# B&R Automation Studio project CoffeeMachine
Automation Studio 4.1.17.113 SP; Default project

## Configuration PP400based

CPU , AutomationRuntime E3.10, Build 4.1.2, Vc V4.15.9, Safety 0.0

### Task classes (Cpu.sw)
```
Cyclic#1:
  mainlogic <- mainlogic.prg
  feeder <- FeederArm.feeder.prg
  conveyor <- ConveyorBelt.conveyor.prg
  heating <- FlowHeater.heating.prg
  brewing <- BrewingAssembly.brewing.prg
Cyclic#4:
  visCtrl <- Visualisation.visCtrl.prg
  visAlarm <- Visualisation.visAlarm.prg
  visTrend <- Visualisation.visTrend.prg
DataObjects: espres <- Recipes.espres.dob, cappu <- Recipes.cappu.dob, regular <- Recipes.regular.dob, Acp10sys, acp10sys
NcDataObjects: motor_offi <- FeederArm.motor_office.dob, motor_sim <- FeederArm.motor_sim.dob, conv_ini <- ConveyorBelt.conv_ini.dob, feed_ini <- FeederArm.feed_ini.dob, acp_err <- FeederArm.acp_err.dob
VcDataObjects: Visu <- Visualisation.Visu.dob
Binaries: vcctext, vcresman, vccovl, vcfile, vcpdpp30, vcdsloc, vcbclass, vcfntttf, vcgclass, vcshared, vcrt, vccbmp, vccbar, vcnet, vccbtn, vcmgr, vctcal, vcptelo, vcalarm, vccnum, vcdsint, Visu02, vccalarm, vcpdvnc, vcpdsw, vccline, vccstr, vcpfpp30, vcctrend, vcclbox, Visu01, vcpfmtcx, Visu03, arialbd, arial, visvc, vcchspot, arialxsr, vcchtml, vcxml, vccslider, vccurl, vccgauge, vcpkat, acp10map, acp10cfg, iomap, arconfig, asfw, sysconf, ashwd, vccshape, arialu_1, vcbmpng, vcpdcx55, vcpfpp, vcptham, ARIAL, ARIALU_1, ARIALBD, Acp10map, Acp10cfg
Libraries: powerlnk, standard, runtime, loopconr, astime, fileio, CoffeeLib, visapi, ashw, asarsdm, dataobj, Acp10_MC, brsystem, sys_lib, Acp10par, NcGlobal
```

### Hardware
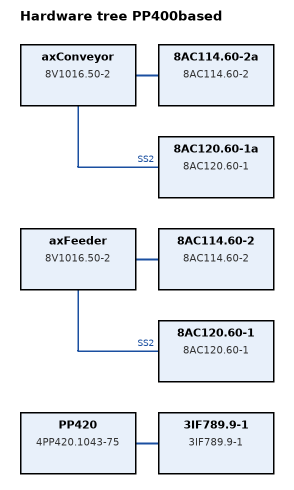
```
3IF789.9-1 : 3IF789.9-1 v1.1.1.0  [SS -> PP420.SS1]
8AC114.60-2 : 8AC114.60-2 v1.0.0.5  [SS -> axFeeder.SS1; PLK1 -> 3IF789.9-1.IF2 (NodeNumber=1)]
8AC114.60-2a : 8AC114.60-2 v1.0.0.5  [SS -> axConveyor.SS1; PLK1 -> 8AC114.60-2.PLK2 (NodeNumber=2)]
8AC120.60-1 : 8AC120.60-1 v1.0.0.2  [SS -> axFeeder.SS2]
8AC120.60-1a : 8AC120.60-1 v1.0.0.2  [SS -> axConveyor.SS2]
axConveyor : 8V1016.50-2 v1.0.0.3
axFeeder : 8V1016.50-2 v1.0.0.3
PP420 : 4PP420.1043-75 v1.0.0.0
  Connector IF5:
    ActivateDevice = 1
    Vnc1
    VncVcObjectName1 = Visu
    VncKeyMappingFile1 = PS2-Keyboard0.dis
    VncAuthentication1 = 1
    VncPasswordViewOnly1 = v
    VncPasswordViewControl1 = c
    VncRefreshRate1 = 100
    VncTitle1 = VNC - B&R Coffee Machine
  BRObjects = 460
  TimerDeviceType = EPLX2X
  TimerDevice = 3IF789.9-1.IF2
  TaskClassIdleTime = 2000
  XLinkUseDefault = 0
  XLinkDuration = 10000
  FileDevice1
  FileDeviceName1 = DISK_C
  FileDevicePath1 = C:\
  EthernetHostName = PP400CoffeeMachine
  ActivateDns = 1
  GetDnsFromDhcp = 2
  VcObjectName = Visu
```

### Acp10cfg.ncc - PP420/Motion/Acp10cfg.ncc
```
NcConfiguration (Version=2.14.0, NcSwId=acp10)
  ACP10CF1_typ:
    cnt_nettrc_rec_drive = 150
    bufsize_trace_upload = 1200
    tc_nc_man_task = Cyclic #1
    glob_pv_as_ncobject = Yes
    network_init:
      ncsw_init_execute = Yes
      automatic_execute = No
      node_nr_warning = Yes
      net_err_before_ncact = Yes
    nettrc:
      enter_parsecrec = Yes
      enter_ncaction = Yes
      save_ring_startidx = No
    plk_if[0]:
      if_name = SL1.SS1.IF2
```

### Acp10map.ncm - PP420/Motion/Acp10map.ncm
```
NcMapping (NcSwId=acp10)
  NcObject axFeeder (ModuleId=axFeeder, Type=ncAXIS, Channel=1, AcoposSimulation=Off, InitParameter=feed_ini, AcoposParameter=motor_sim, AdditionalData=PLCopen_ModPos="36000,100", Disabled=FALSE, ModuleDisabled=FALSE)
  NcObject axConveyor (ModuleId=axConveyor, Type=ncAXIS, Channel=1, AcoposSimulation=Off, InitParameter=conv_ini, AcoposParameter=motor_sim, AdditionalData=PLCopen_ModPos="8388608,100", Disabled=FALSE, ModuleDisabled=FALSE)
  NcObject SL1.SS1.IF2.ST2.VAxis1 (ModuleId=axConveyor, Type=ncV_AXIS, Channel=1, Disabled=TRUE, ModuleDisabled=FALSE)
  NcObject SL1.SS1.IF2.ST1.VAxis1 (ModuleId=axFeeder, Type=ncV_AXIS, Channel=1, Disabled=TRUE, ModuleDisabled=FALSE)
```

## Configuration PP400mcSim

CPU , AutomationRuntime E3.10, Build 4.1.2, Vc V4.15.9, Safety 0.0

### Task classes (Cpu.sw)
```
Cyclic#1 (cycle 2000 us, tolerance 0 us):
  mainlogic <- mainlogic.prg
  feeder <- FeederArm.feeder.prg
  conveyor <- ConveyorBelt.conveyor.prg
  heating <- FlowHeater.heating.prg
  brewing <- BrewingAssembly.brewing.prg
Cyclic#4 (cycle 100000 us, tolerance 100000 us):
  visCtrl <- Visualisation.visCtrl.prg
  visAlarm <- Visualisation.visAlarm.prg
  visTrend <- Visualisation.visTrend.prg
DataObjects: espres <- Recipes.espres.dob, cappu <- Recipes.cappu.dob, regular <- Recipes.regular.dob, Acp10sys
NcDataObjects: acp_err <- FeederArm.acp_err.dob, motor_sim <- FeederArm.motor_sim.dob, motor_offi <- FeederArm.motor_office.dob, conv_ini <- ConveyorBelt.conv_ini.dob, feed_ini <- FeederArm.feed_ini.dob
VcDataObjects: Visu <- Visualisation.Visu.dob
Binaries: ARIALBD, ARIALU_1, ARIAL, vcptham, vcpfpp, vcpdcx55, vcbmpng, arialu_1, vcpkat, Acp10map, Acp10cfg, vccshape, ashwd, sysconf, asfw, arconfig, iomap, acp10cfg, acp10map, vccgauge, vccslider, vccurl, vcxml, vcchtml, arialxsr, visvc, arial, arialbd, Visu03, vcpfmtcx, Visu01, vcclbox, vcctrend, vcpfpp30, vccstr, vccline, vcpdsw, vcpdvnc, vccalarm, Visu02, vcdsint, vccnum, vcalarm, vcptelo, vctcal, vcmgr, vccbtn, vcnet, vccbar, vccbmp, vcrt, vcshared, vcgclass, vcfntttf, vcbclass, vcdsloc, vcpdpp30, vcfile, vccovl, vcresman, vcctext, vcchspot
Libraries: sys_lib, brsystem, FileIO, AsTime, CoffeeLib, Acp10par, NcGlobal, AsArSdm, Acp10sdc, ashw, visapi, dataobj, loopconr, runtime, standard, powerlnk
```

### Hardware
```
PP420 : 4PP420.1043-75 v1.0.0.0
  Connector IF5:
    ActivateDevice = 1
    Vnc1
    VncVcObjectName1 = Visu
    VncAuthentication1 = 1
    VncPasswordViewOnly1 = v
    VncPasswordViewControl1 = c
    VncTitle1 = VNC - B&R Coffee Machine
  BRObjects = 450
  Cyclic1Duration = 2000
  Cyclic1Tolerance = 0
  Cyclic2Duration = 20000
  Cyclic2Tolerance = 20000
  Cyclic3Duration = 50000
  Cyclic3Tolerance = 50000
  Cyclic4Duration = 100000
  Cyclic4Tolerance = 100000
  Cyclic5Duration = 200000
  Cyclic5Tolerance = 200000
  Cyclic6Duration = 500000
  Cyclic6Tolerance = 500000
  Cyclic7Duration = 1000000
  Cyclic7Tolerance = 1000000
  Cyclic8Duration = 10000
  Cyclic8Tolerance = 30000000
  EthernetHostName = PP400CoffeeMachine
  ActivateDns = 1
  GetDnsFromDhcp = 2
  VcObjectName = Visu
```

## Configuration PP500mcSim

CPU , AutomationRuntime G4.09, Build 4.1.2, Vc V4.15.9, Safety 0.0

### Task classes (Cpu.sw)
```
Cyclic#1 (cycle 2000 us, tolerance 0 us):
  mainlogic <- mainlogic.prg
  feeder <- FeederArm.feeder.prg
  conveyor <- ConveyorBelt.conveyor.prg
  brewing <- BrewingAssembly.brewing.prg
  heating <- FlowHeater.heating.prg
Cyclic#4 (cycle 100000 us, tolerance 100000 us):
  visCtrl <- Visualisation.visCtrl.prg
  visAlarm <- Visualisation.visAlarm.prg
  visTrend <- Visualisation.visTrend.prg
DataObjects: cappu <- Recipes.cappu.dob, regular <- Recipes.regular.dob, espres <- Recipes.espres.dob, Acp10sys
NcDataObjects: acp_err <- FeederArm.acp_err.dob, motor_sim <- FeederArm.motor_sim.dob, motor_offi <- FeederArm.motor_office.dob, feed_ini <- FeederArm.feed_ini.dob, conv_ini <- ConveyorBelt.conv_ini.dob
VcDataObjects: VisuW <- Visualisation.VisuW.dob
Binaries: vccalarm, vcclbox, vcctext, vcrt, VisuW03, vccnum, vcchspot, vccbar, vccurl, vcchtml, vcfile, arialxsr, vcpdsw, vccbmp, vcshared, vcctrend, vcfntttf, vcgclass, vccovl, arialbd, vcdsint, vccslider, vcalarm, vccline, vcresman, vcdsloc, vccbtn, vccstr, vcbclass, vcxml, VisuW02, arial, vccdt, vccgauge, vcmgr, vcptelo, vcpdihd, vcpfpp50, vcpdi855, visvc, vccshape, VisuW01, vcpdi815, vcpfmtcx, vctcal, Acp10cfg, Acp10map, iomap, asfw, ashwd, sysconf, arconfig
Libraries: Acp10sdc, standard, loopconr, astime, runtime, powerlnk, CoffeeLib, Acp10par, AsArSdm, NcGlobal, brsystem, sys_lib, Acp10man, fileio, visapi, dataobj, acp10_mc
```

### Hardware
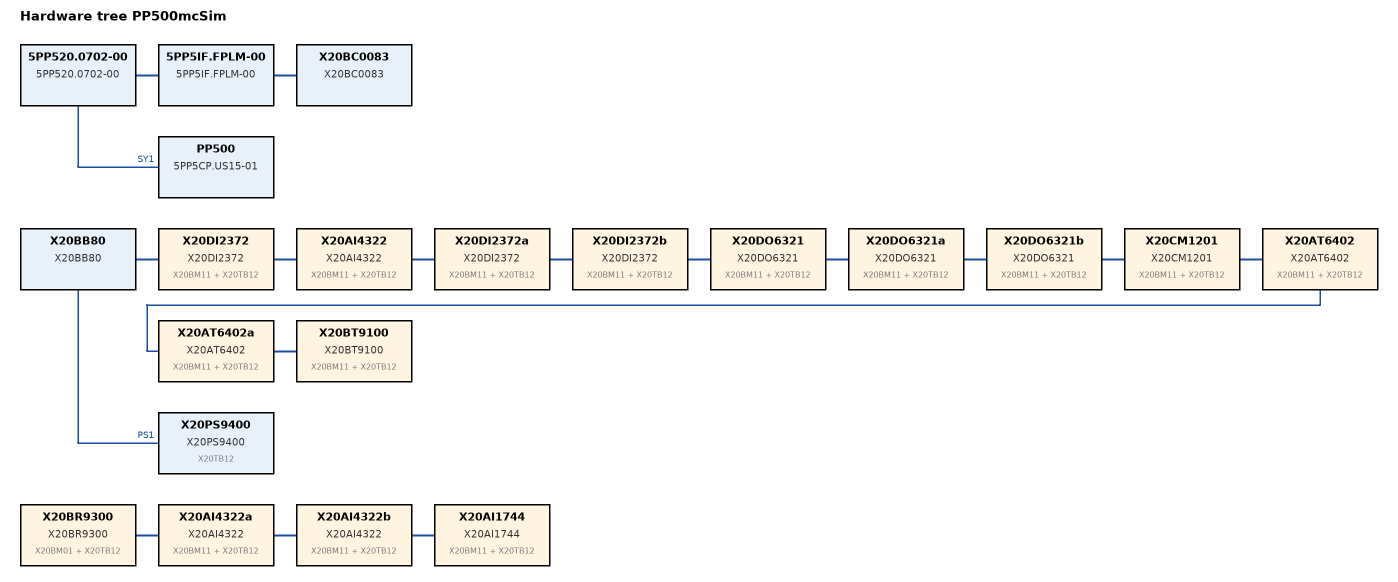
```
5PP520.0702-00 : 5PP520.0702-00 v2.0.1.2
  Connector IF3:
    ActivateDevice = 1
    EthInterfaceRedundant = 0
    HostName = pp500coffeemachine
  VcObjectName = VisuW
5PP5IF.FPLM-00 : 5PP5IF.FPLM-00 v2.2.0.0  [SL -> 5PP520.0702-00.SL1]
  Connector IF1:
    EplEthInterfaceRedundant = 0
  Supervision = off
PP500 : 5PP5CP.US15-01 v2.0.3.2  [SY -> 5PP520.0702-00.SY1]
  PreserveNonVolatileSystemSettings = 0
  BRObjects = 450
  Cyclic1Duration = 2000
  Cyclic1Tolerance = 0
  Cyclic2Duration = 20000
  Cyclic2Tolerance = 20000
  Cyclic3Duration = 50000
  Cyclic3Tolerance = 50000
  Cyclic4Duration = 100000
  Cyclic4Tolerance = 100000
  Cyclic5Duration = 200000
  Cyclic5Tolerance = 200000
  Cyclic6Duration = 500000
  Cyclic6Tolerance = 500000
  Cyclic7Duration = 1000000
  Cyclic7Tolerance = 1000000
  Cyclic8Duration = 10000
  Cyclic8Tolerance = 30000000
  EthernetHostName = brautomation
  ActivateDns = 1
X20AI1744 : X20AI1744 v1.3.0.1  [SS1 -> X20TB12o.SS; SL -> X20BM11m.SL1]
  Supervision = off
X20AI4322 : X20AI4322 v1.0.0.1  [SS1 -> X20TB12b.SS; SL -> X20BM11a.SL1]
  Supervision = off
X20AI4322a : X20AI4322 v1.0.0.1  [SS1 -> X20TB12m.SS; SL -> X20BM11k.SL1]
  Supervision = off
X20AI4322b : X20AI4322 v1.0.0.1  [SS1 -> X20TB12n.SS; SL -> X20BM11l.SL1]
  Supervision = off
X20AT6402 : X20AT6402 v1.0.2.2  [SS1 -> X20TB12i.SS; SL -> X20BM11h.SL1]
  Supervision = off
X20AT6402a : X20AT6402 v1.0.2.2  [SS1 -> X20TB12j.SS; SL -> X20BM11i.SL1]
  Supervision = off
X20BB80 : X20BB80 v1.0.0.2
X20BC0083 : X20BC0083 v2.0.0.0  [PLK1 -> 5PP5IF.FPLM-00.IF1 (NodeNumber=1); SL -> X20BB80.SL1]
  Supervision = off
X20BM01 : X20BM01 v1.0.0.1
X20BM11 : X20BM11 v1.0.0.0  [X2X1 -> X20BB80.IF1]
X20BM11a : X20BM11 v1.0.0.0  [X2X1 -> X20BM11.X2X2]
X20BM11b : X20BM11 v1.0.0.0  [X2X1 -> X20BM11a.X2X2]
X20BM11c : X20BM11 v1.0.0.0  [X2X1 -> X20BM11b.X2X2]
X20BM11d : X20BM11 v1.0.0.0  [X2X1 -> X20BM11c.X2X2]
X20BM11e : X20BM11 v1.0.0.0  [X2X1 -> X20BM11d.X2X2]
X20BM11f : X20BM11 v1.0.0.0  [X2X1 -> X20BM11e.X2X2]
X20BM11g : X20BM11 v1.0.0.0  [X2X1 -> X20BM11f.X2X2]
X20BM11h : X20BM11 v1.0.0.0  [X2X1 -> X20BM11g.X2X2]
X20BM11i : X20BM11 v1.0.0.0  [X2X1 -> X20BM11h.X2X2]
X20BM11j : X20BM11 v1.0.0.0  [X2X1 -> X20BM11i.X2X2]
X20BM11k : X20BM11 v1.0.0.0  [X2X1 -> X20BM01.X2X2]
X20BM11l : X20BM11 v1.0.0.0  [X2X1 -> X20BM11k.X2X2]
X20BM11m : X20BM11 v1.0.0.0  [X2X1 -> X20BM11l.X2X2]
X20BR9300 : X20BR9300 v1.0.2.4  [SS1 -> X20TB12l.SS; SL -> X20BM01.SL1; X2X1 -> X20BT9100.X2X1]
  Supervision = off
X20BT9100 : X20BT9100 v1.0.2.3  [SS1 -> X20TB12k.SS; SL -> X20BM11j.SL1]
  Supervision = off
X20CM1201 : X20CM1201 v1.0.0.0  [SS1 -> X20TB12h.SS; SL -> X20BM11g.SL1]
  Supervision = off
X20DI2372 : X20DI2372 v1.0.1.0  [SS1 -> X20TB12a.SS; SL -> X20BM11.SL1]
  Supervision = off
X20DI2372a : X20DI2372 v1.0.1.0  [SS1 -> X20TB12c.SS; SL -> X20BM11b.SL1]
  Supervision = off
X20DI2372b : X20DI2372 v1.0.1.0  [SS1 -> X20TB12d.SS; SL -> X20BM11c.SL1]
  Supervision = off
X20DO6321 : X20DO6321 v1.0.1.0  [SS1 -> X20TB12e.SS; SL -> X20BM11d.SL1]
  Supervision = off
X20DO6321a : X20DO6321 v1.0.1.0  [SS1 -> X20TB12f.SS; SL -> X20BM11e.SL1]
  Supervision = off
X20DO6321b : X20DO6321 v1.0.1.0  [SS1 -> X20TB12g.SS; SL -> X20BM11f.SL1]
  Supervision = off
X20PS9400 : X20PS9400 v1.0.2.0  [SS1 -> X20TB12.SS; PS -> X20BB80.PS1]
  Supervision = off
X20TB12 : X20TB12 v1.0.0.0
X20TB12a : X20TB12 v1.0.0.0
X20TB12b : X20TB12 v1.0.0.0
X20TB12c : X20TB12 v1.0.0.0
X20TB12d : X20TB12 v1.0.0.0
X20TB12e : X20TB12 v1.0.0.0
X20TB12f : X20TB12 v1.0.0.0
X20TB12g : X20TB12 v1.0.0.0
X20TB12h : X20TB12 v1.0.0.0
X20TB12i : X20TB12 v1.0.0.0
X20TB12j : X20TB12 v1.0.0.0
X20TB12k : X20TB12 v1.0.0.0
X20TB12l : X20TB12 v1.0.0.0
X20TB12m : X20TB12 v1.0.0.0
X20TB12n : X20TB12 v1.0.0.0
X20TB12o : X20TB12 v1.0.0.0
```

### Acp10cfg.ncc - PP500/Motion/Acp10cfg.ncc
```
NcConfiguration (Version=2.14.0, NcSwId=acp10)
  ACP10CF1_typ:
    cnt_nettrc_rec_drive = 150
    bufsize_trace_upload = 1200
    tc_nc_man_task = Cyclic #1
    glob_pv_as_ncobject = Yes
    network_init:
      ncsw_init_execute = Yes
      automatic_execute = No
      node_nr_warning = Yes
      net_err_before_ncact = Yes
    nettrc:
      enter_parsecrec = Yes
      enter_ncaction = Yes
    sdc_if[0]:
      if_name = SDC_IF1
```

### Acp10map.ncm - PP500/Motion/Acp10map.ncm
```
NcMapping (NcSwId=acp10)
  NcObject axFeeder (ModuleAddress=SDC_IF1.ST1, InterfaceType=SDC, Type=ncAXIS, Channel=1, AcoposSimulation=Off, InitParameter=feed_ini, AcoposParameter=motor_sim, AdditionalData=PLCopen_ModPos="36000,100", Disabled=FALSE, ModuleDisabled=FALSE)
  NcObject axConveyor (ModuleAddress=SDC_IF1.ST2, InterfaceType=SDC, Type=ncAXIS, Channel=1, AcoposSimulation=Off, InitParameter=conv_ini, AcoposParameter=motor_sim, AdditionalData=PLCopen_ModPos="8388608,100", Disabled=FALSE, ModuleDisabled=FALSE)
```

## Configuration PP65mcSim

CPU 4PP065.0571-P74, AutomationRuntime E3.10, Build 4.1.2, Vc V4.15.9, Safety 0.0

### Hardware
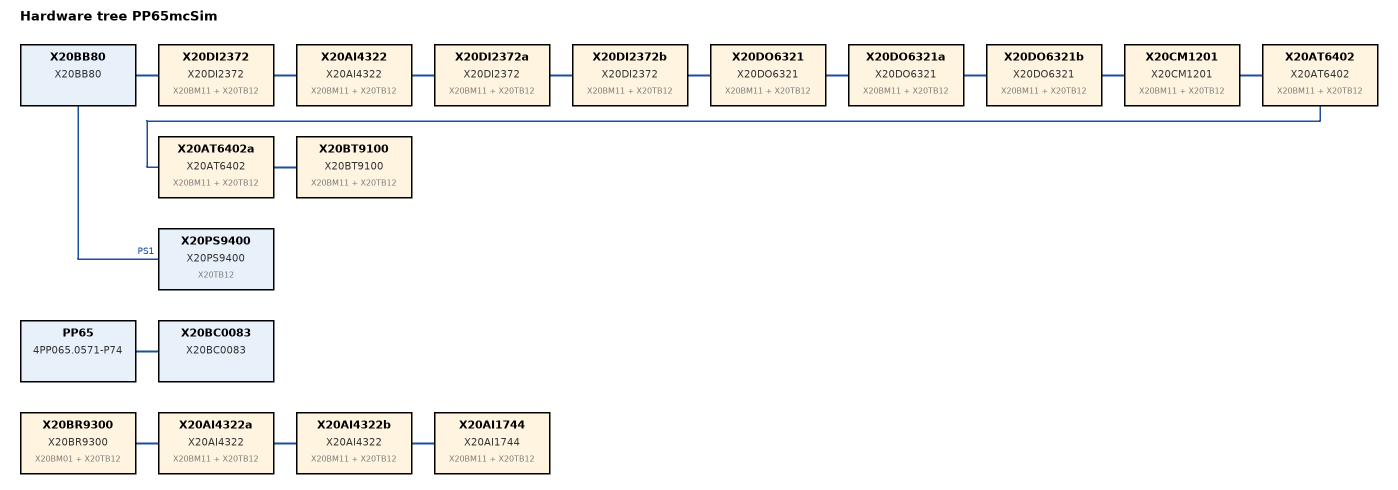
```
PP65 : 4PP065.0571-P74 v1.0.2.1
  Connector IF4:
    EplInterfaceRedundant = 0
    EplEthInterfaceRedundant = 0
  Connector IF5:
    ActivateDevice = 1
    HostName = pp500coffeemachine
    Mode = Manual
    InternetAddress = 10.49.40.222
    SubnetMask = 255.255.255.0
  PreserveNonVolatileSystemSettings = 0
  BRObjects = 450
  Cyclic1Duration = 10000
  Cyclic1Tolerance = 10000
  Cyclic2Duration = 20000
  Cyclic2Tolerance = 20000
  Cyclic3Duration = 50000
  Cyclic3Tolerance = 50000
  Cyclic4Duration = 100000
  Cyclic4Tolerance = 100000
  Cyclic5Duration = 200000
  Cyclic5Tolerance = 200000
  Cyclic6Duration = 500000
  Cyclic6Tolerance = 500000
  Cyclic7Duration = 1000000
  Cyclic7Tolerance = 1000000
  Cyclic8Duration = 10000
  Cyclic8Tolerance = 30000000
  EthernetHostName = brautomation
  ActivateDns = 1
X20AI1744 : X20AI1744 v1.3.0.1  [SS1 -> X20TB12o.SS; SL -> X20BM11m.SL1]
  Supervision = off
X20AI4322 : X20AI4322 v1.0.0.1  [SS1 -> X20TB12b.SS; SL -> X20BM11a.SL1]
  Supervision = off
X20AI4322a : X20AI4322 v1.0.0.1  [SS1 -> X20TB12m.SS; SL -> X20BM11k.SL1]
  Supervision = off
X20AI4322b : X20AI4322 v1.0.0.1  [SS1 -> X20TB12n.SS; SL -> X20BM11l.SL1]
  Supervision = off
X20AT6402 : X20AT6402 v1.0.2.2  [SS1 -> X20TB12i.SS; SL -> X20BM11h.SL1]
  Supervision = off
X20AT6402a : X20AT6402 v1.0.2.2  [SS1 -> X20TB12j.SS; SL -> X20BM11i.SL1]
  Supervision = off
X20BB80 : X20BB80 v1.0.0.2
X20BC0083 : X20BC0083 v2.0.0.0  [PLK1 -> PP65.IF4 (NodeNumber=1); SL -> X20BB80.SL1]
  Supervision = off
X20BM01 : X20BM01 v1.0.0.1
X20BM11 : X20BM11 v1.0.0.0  [X2X1 -> X20BB80.IF1]
X20BM11a : X20BM11 v1.0.0.0  [X2X1 -> X20BM11.X2X2]
X20BM11b : X20BM11 v1.0.0.0  [X2X1 -> X20BM11a.X2X2]
X20BM11c : X20BM11 v1.0.0.0  [X2X1 -> X20BM11b.X2X2]
X20BM11d : X20BM11 v1.0.0.0  [X2X1 -> X20BM11c.X2X2]
X20BM11e : X20BM11 v1.0.0.0  [X2X1 -> X20BM11d.X2X2]
X20BM11f : X20BM11 v1.0.0.0  [X2X1 -> X20BM11e.X2X2]
X20BM11g : X20BM11 v1.0.0.0  [X2X1 -> X20BM11f.X2X2]
X20BM11h : X20BM11 v1.0.0.0  [X2X1 -> X20BM11g.X2X2]
X20BM11i : X20BM11 v1.0.0.0  [X2X1 -> X20BM11h.X2X2]
X20BM11j : X20BM11 v1.0.0.0  [X2X1 -> X20BM11i.X2X2]
X20BM11k : X20BM11 v1.0.0.0  [X2X1 -> X20BM01.X2X2]
X20BM11l : X20BM11 v1.0.0.0  [X2X1 -> X20BM11k.X2X2]
X20BM11m : X20BM11 v1.0.0.0  [X2X1 -> X20BM11l.X2X2]
X20BR9300 : X20BR9300 v1.0.2.4  [SS1 -> X20TB12l.SS; SL -> X20BM01.SL1; X2X1 -> X20BT9100.X2X1]
  Supervision = off
X20BT9100 : X20BT9100 v1.0.2.3  [SS1 -> X20TB12k.SS; SL -> X20BM11j.SL1]
  Supervision = off
X20CM1201 : X20CM1201 v1.0.0.0  [SS1 -> X20TB12h.SS; SL -> X20BM11g.SL1]
  Supervision = off
X20DI2372 : X20DI2372 v1.0.1.0  [SS1 -> X20TB12a.SS; SL -> X20BM11.SL1]
  Supervision = off
X20DI2372a : X20DI2372 v1.0.1.0  [SS1 -> X20TB12c.SS; SL -> X20BM11b.SL1]
  Supervision = off
X20DI2372b : X20DI2372 v1.0.1.0  [SS1 -> X20TB12d.SS; SL -> X20BM11c.SL1]
  Supervision = off
X20DO6321 : X20DO6321 v1.0.1.2  [SS1 -> X20TB12e.SS; SL -> X20BM11d.SL1]
  Supervision = off
X20DO6321a : X20DO6321 v1.0.1.2  [SS1 -> X20TB12f.SS; SL -> X20BM11e.SL1]
  Supervision = off
X20DO6321b : X20DO6321 v1.0.1.2  [SS1 -> X20TB12g.SS; SL -> X20BM11f.SL1]
  Supervision = off
X20PS9400 : X20PS9400 v1.0.2.0  [SS1 -> X20TB12.SS; PS -> X20BB80.PS1]
  Supervision = off
X20TB12 : X20TB12 v1.0.0.0
X20TB12a : X20TB12 v1.0.0.0
X20TB12b : X20TB12 v1.0.0.0
X20TB12c : X20TB12 v1.0.0.0
X20TB12d : X20TB12 v1.0.0.0
X20TB12e : X20TB12 v1.0.0.0
X20TB12f : X20TB12 v1.0.0.0
X20TB12g : X20TB12 v1.0.0.0
X20TB12h : X20TB12 v1.0.0.0
X20TB12i : X20TB12 v1.0.0.0
X20TB12j : X20TB12 v1.0.0.0
X20TB12k : X20TB12 v1.0.0.0
X20TB12l : X20TB12 v1.0.0.0
X20TB12m : X20TB12 v1.0.0.0
X20TB12n : X20TB12 v1.0.0.0
X20TB12o : X20TB12 v1.0.0.0
```

## Configuration Simulation

CPU , AutomationRuntime G4.09, Build 4.1.2, Vc V4.15.9, Safety 0.0

### Task classes (AppMo.sw)
```
Cyclic#1 (cycle 10000 us, tolerance 0 us):
  myApptask1 <- myAppMod1.myApptask1.prg
```

### Task classes (Cpu.sw)
```
Cyclic#1 (cycle 10000 us, tolerance 0 us):
  mainlogic <- mainlogic.prg
  feeder <- FeederArm.feeder.prg
  conveyor <- ConveyorBelt.conveyor.prg
  brewing <- BrewingAssembly.brewing.prg
  heating <- FlowHeater.heating.prg
Cyclic#2:
  visCtrl <- Visualisation.visCtrl.prg
Cyclic#4:
  visAlarm <- Visualisation.visAlarm.prg
  visTrend <- Visualisation.visTrend.prg
  NewProgram <- NewProgram.prg
  myProg <- myProg.prg
DataObjects: regular <- Recipes.regular.dob, cappu <- Recipes.cappu.dob, espres <- Recipes.espres.dob, empty1 <- Recipes.empty1.dob, object2 <- Recipes.object2.dob, data <- data.dob
NcDataObjects: acp_err <- FeederArm.acp_err.dob, motor_sim <- FeederArm.motor_sim.dob, motor_offi <- FeederArm.motor_office.dob, feed_ini <- FeederArm.feed_ini.dob, conv_ini <- ConveyorBelt.conv_ini.dob, cnc1 <- cnc1.dob, cnc2 <- cnc2.dob, cnc3 <- cnc3.dob
VcDataObjects: Visu <- Visualisation.Visu.dob
Binaries: vccslider, vccurl, vcxml, vcchtml, arialxsr, vcchspot, vcctext, vcresman, vccovl, vcfile, vcdsloc, vcbclass, vcfntttf, vccstr, vcgclass, vcshared, vcrt, vccbmp, vccbar, vccbtn, vcmgr, vctcal, visvc, vcalarm, vccnum, vcdsint, vccalarm, vccline, vcpdvnc, vcpdsw, vcnet, vcctrend, vcclbox, vcpfar00, Visu01, Visu02, Visu03, vccgauge, vccshape, vccdt, arial, arialbd, acp10cfg, acp10map, arconfig, asfw, ashwd, sysconf, iomap, arialu_1, vcbmpng, ARIALU_1, Acp10map, Acp10cfg, ARIALBD, ARIAL
Libraries: AsTime, CoffeeLib, FileIO, NcGlobal, Acp10par, Convert, Visapi, AsArSdm, Runtime, operator, standard, dataobj, powerlnk, brsystem, sys_lib, Acp10man, Acp10sim, Acp10_MC, Acp10sdc, AsArProf, loopconr, vcscrsht
```

### Hardware
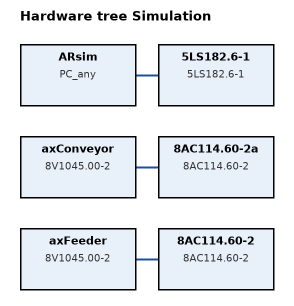
```
5LS182.6-1 : 5LS182.6-1 v1.2.2.1  [SL -> ARsim.SL1]
8AC114.60-2 : 8AC114.60-2 v1.0.0.5  [SS -> axFeeder.SS1; PLK1 -> 5LS182.6-1.IF1 (NodeNumber=1)]
8AC114.60-2a : 8AC114.60-2 v1.0.0.5  [SS -> axConveyor.SS1; PLK1 -> 8AC114.60-2.PLK2 (NodeNumber=2)]
ARsim : PC_any v1.1.0.0 (OrderNumber=PC)
  Connector IF3:
    Vnc1
    VncVcObjectName1 = Visu
    VncAuthentication1 = 1
    VncPasswordViewOnly1 = v
    VncPasswordViewControl1 = c
    VncRefreshRate1 = 200
    VncTitle1 = VNC - B&R Coffee Machine
  PreserveNonVolatileSystemSettings = 0
  BRObjects = 450
  XLinkUseDefault = 0
  Cyclic1Duration = 10000
  Cyclic1Tolerance = 0
  EthernetHostName = AR000CoffeeMachine
  ActivateOpcUa = 1
axConveyor : 8V1045.00-2 v1.0.0.2
  Simulate = standard
axFeeder : 8V1045.00-2 v1.0.0.2
  Simulate = standard
```

### Acp10cfg.ncc - ARsim/Motion/Acp10cfg.ncc
```
NcConfiguration (Version=2.37.0, NcSwId=Acp10)
  ACP10CF1_typ:
    cnt_nettrc_rec_drive = 150
    bufsize_trace_upload = 1200
    tc_nc_man_task = Cyclic #1
    glob_pv_as_ncobject = Yes
    ncsys_dl_broadcast = Yes
    ncsys_dl_acp_reset = Yes
    network_init:
      ncsw_init_execute = Yes
      automatic_execute = No
      node_nr_warning = Yes
      net_err_before_ncact = Yes
    nettrc:
      enter_parsecrec = Yes
      enter_ncaction = Yes
      save_ring_startidx = No
    plk_if[0]:
      if_name = SL1.IF1
      tc_CycDat_PLCopen = Task class for NC Manager task
      mc_broadcast_extdat = No
```

## Logical view

Binary libraries used (declarations not repeated): Convert, Runtime, sys_lib, brsystem, Standard, AsString, DataObj, FileIO, operator, AsTime, LoopConR 2.68.0, Visapi, AsArSdm, AsArProf, Acp10man 2.45.1, Acp10par 2.45.1, NcGlobal 2.45.1, Acp10sdc 2.45.1, Acp10sim 2.45.1, Acp10_MC 2.45.1

### Global.var - Global Variables
```iecst
(********************************************************************
 * COPYRIGHT -- B&R
 ********************************************************************
 * File: Global.var
 * Author: B&R
 * Created: June 06, 2007
 ********************************************************************
 * Global variables of project coffee
 ********************************************************************)
VAR
	axFeeder : ACP10AXIS_typ; (*axis information of feeder*)
	axConveyor : ACP10AXIS_typ; (*axis information of conveyor*)
	doCupPull : BOOL := FALSE; (*pulls cup out of storage*)
	gMainLogic : main_typ; (*info structure of main logic*)
	gFeeder : feeder_typ := (0); (*info structure of feeder*)
	gBrewing : brewing_typ := (0); (*info structure of brewing assembly*)
	doDoseMilk : BOOL := FALSE; (*doser: milk*)
	doDoseSugar : BOOL := FALSE; (*doser: sugar*)
	doDoseCoffee : BOOL := FALSE; (*doser: coffee*)
	gConveyor : conveyor_typ := (0);
	gHeating : heating_typ := (0); (*info structure of heating*)
	doPumpWater : BOOL := FALSE; (*water pump*)
	aoHeating : INT := 0; (*heating control*)
	atWaterTemp : INT := 0; (*actual temperature of water*)
	diStartCoffee : BOOL := FALSE; (*start making coffee*)
	gActConveyorVelocity : REAL; (*actual conveyor velocity*)
	gActFeederVelocity : REAL; (*actual feeder velocity*)
	gActFeederPosition : REAL; (*actual feeder position*)
	gActConveyorPosition : REAL; (*actual conveyor position*)
END_VAR
```

### Program Logical/mainlogic (IEC, version 1.00.0) - Main Logic Control

#### MainLogicCyclic.cfc - Cyclic code
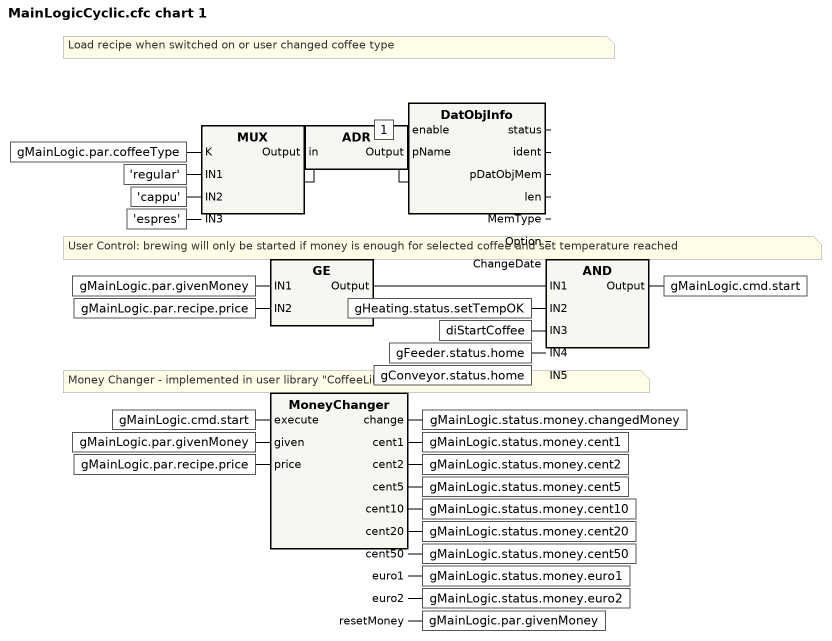
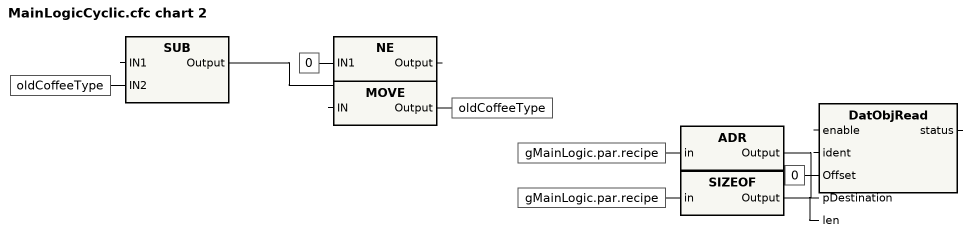
Diagram, in the editor's own instruction-list form stored in the file:
```il
PROGRAM _CYCLIC
(* Load recipe when switched on or user changed coffee type *)
(* User Control: brewing will only be started if money is enough for selected coffee and set temperature reached *)
(* Money Changer - implemented in user library "CoffeeLib" *)
VAR
	zz0000FCT_10_1_MUX_Output : ANY;
	zz0000FCT_10_1_GE_Output : BOOL;
	zz0000FB_10_1_MoneyChanger : MoneyChanger;
	zz0000FCT_10_1_ADR_Output : UDINT;
	zz0000FB_10_1_DatObjInfo : DatObjInfo;
	zz0000FCT_10_55_1_SUB_Output : ANY;
	zz0000FCT_10_55_1_NE_Output : BOOL;
	zz0000FCT_10_2_ADR_Output : UDINT;
	zz0000FCT_10_1_SIZEOF_Output : UDINT;
	zz0000FB_10_1_DatObjRead : DatObjRead;
END_VAR

LD gMainLogic.par.coffeeType
MUX 'regular', 'cappu', 'espres'
ST zz0000FCT_10_1_MUX_Output
LD gMainLogic.par.givenMoney
GE gMainLogic.par.recipe.price
ST zz0000FCT_10_1_GE_Output
LD gMainLogic.cmd.start
ST zz0000FB_10_1_MoneyChanger.execute
LD gMainLogic.par.givenMoney
ST zz0000FB_10_1_MoneyChanger.given
LD gMainLogic.par.recipe.price
ST zz0000FB_10_1_MoneyChanger.price
CAL zz0000FB_10_1_MoneyChanger
LD zz0000FB_10_1_MoneyChanger.change
ST gMainLogic.status.money.changedMoney
LD zz0000FB_10_1_MoneyChanger.cent1
ST gMainLogic.status.money.cent1
LD zz0000FB_10_1_MoneyChanger.cent2
ST gMainLogic.status.money.cent2
LD zz0000FB_10_1_MoneyChanger.cent5
ST gMainLogic.status.money.cent5
LD zz0000FB_10_1_MoneyChanger.cent10
ST gMainLogic.status.money.cent10
LD zz0000FB_10_1_MoneyChanger.cent20
ST gMainLogic.status.money.cent20
LD zz0000FB_10_1_MoneyChanger.cent50
ST gMainLogic.status.money.cent50
LD zz0000FB_10_1_MoneyChanger.euro1
ST gMainLogic.status.money.euro1
LD zz0000FB_10_1_MoneyChanger.euro2
ST gMainLogic.status.money.euro2
LD zz0000FB_10_1_MoneyChanger.resetMoney
ST gMainLogic.par.givenMoney
LD zz0000FCT_10_1_MUX_Output
ADR
ST zz0000FCT_10_1_ADR_Output
LD 1
ST zz0000FB_10_1_DatObjInfo.enable
LD zz0000FCT_10_1_ADR_Output
ST zz0000FB_10_1_DatObjInfo.pName
CAL zz0000FB_10_1_DatObjInfo
LD zz0000FCT_10_1_GE_Output
AND gHeating.status.setTempOK
AND diStartCoffee
AND gFeeder.status.home
AND gConveyor.status.home
ST gMainLogic.cmd.start
LD gMainLogic.par.coffeeType
SUB oldCoffeeType
ST zz0000FCT_10_55_1_SUB_Output
LD 0
NE zz0000FCT_10_55_1_SUB_Output
ST zz0000FCT_10_55_1_NE_Output
LD gMainLogic.par.coffeeType
MOVE
ST oldCoffeeType
LD gMainLogic.par.recipe
ADR
ST zz0000FCT_10_2_ADR_Output
LD gMainLogic.par.recipe
SIZEOF
ST zz0000FCT_10_1_SIZEOF_Output
LD zz0000FCT_10_55_1_NE_Output
ST zz0000FB_10_1_DatObjRead.enable
LD zz0000FB_10_1_DatObjInfo.ident
ST zz0000FB_10_1_DatObjRead.ident
LD 0
ST zz0000FB_10_1_DatObjRead.Offset
LD zz0000FCT_10_2_ADR_Output
ST zz0000FB_10_1_DatObjRead.pDestination
LD zz0000FCT_10_1_SIZEOF_Output
ST zz0000FB_10_1_DatObjRead.len
CAL zz0000FB_10_1_DatObjRead

END_PROGRAM
```

#### MainLogicInit.cfc
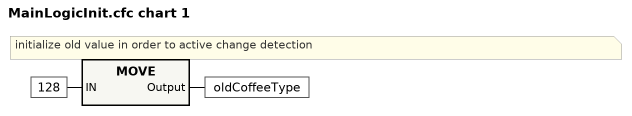
Diagram, in the editor's own instruction-list form stored in the file:
```il
PROGRAM _INIT
(* initialize old value in order to active change detection *)

LD  128
MOVE
ST oldCoffeeType

END_PROGRAM
```

#### mainlogic.var - Local variables
```iecst
(********************************************************************
 * COPYRIGHT -- B&R
 ********************************************************************
 * Package: mainlogic
 * File: mainlogic.var
 * Author: B&R
 * Created: June 18, 2007
 *******************************************************************)
VAR
	oldCoffeeType : SINT := 0;
END_VAR
```

### Package Logical/ConveyorBelt - Conveyor Control

### Data object Logical/ConveyorBelt/conv_ini (Ax) - Conveyor axis configuration

#### conv_ini.ax
```
InitParameter (Version=2.28.2, NcSwId=ACP10)
  ACP10AXIS_typ:
    dig_in:
      level:
        reference = ncACTIV_HI
        pos_hw_end = ncACTIV_HI
        neg_hw_end = ncACTIV_HI
        trigger1 = ncACTIV_HI
        trigger2 = ncACTIV_HI
    encoder_if:
      parameter:
        count_dir = ncSTANDARD
        scaling:
          load:
            units = 5000
            rev_motor = 10
    limit:
      parameter:
        v_pos = 10000
        v_neg = 10000
        a1_pos = 50000
        a2_pos = 50000
        a1_neg = 50000
        a2_neg = 50000
        t_jolt = 0.05
        t_in_pos = 0
        pos_sw_end = 8388607
        neg_sw_end = -8388608
        ds_warning = 500
        ds_stop = 1000
        a_stop = 1e+030
        dv_stop = 0
        dv_stop_mode = ncOFF
    controller:
      mode = ncPOSITION
      position:
        kv = 50
        tn = 0
        t_predict = 0.0008
        t_total = 0.0008
        p_max = 10000
        i_max = 0
      speed:
        kv = 2
        tn = 0
        t_filter = 0
        isq_filter1:
          type = ncOFF
          a0 = 0
          a1 = 0
          b0 = 0
          b1 = 0
          b2 = 0
          c0_par_id = 0
          c1_par_id = 0
        isq_filter2:
          type = ncOFF
          a0 = 0
          a1 = 0
          b0 = 0
          b1 = 0
          b2 = 0
          c0_par_id = 0
          c1_par_id = 0
        isq_filter3:
          type = ncOFF
          a0 = 0
          a1 = 0
          b0 = 0
          b1 = 0
          b2 = 0
          c0_par_id = 0
          c1_par_id = 0
      uf:
        type = ncLINEAR
        auto_config = ncMOTOR_PAR
        u0 = 0
        un = 0
        fn = 50
        k_f_slip = 0
      ff:
        torque_load = 0
        torque_pos = 0
        torque_neg = 0
        kv_torque = 0
        inertia = 0
        t_filter_a = 0
    move:
      stop:
        parameter[0]:
          decel_ramp = ncA_LIMIT
          controller = ncON
        parameter[1]:
          decel_ramp = ncA_LIMIT
          controller = ncON
        parameter[2]:
          decel_ramp = ncA_LIMIT
          controller = ncON
        parameter[3]:
          decel_ramp = ncA_LIMIT
          controller = ncON
        quickstop:
          decel_ramp = ncA_LIMIT
        drive_error:
          decel_ramp = ncA_LIMIT
      homing:
        parameter:
          s = 0
          v_switch = 5000
          v_trigger = 500
          a = 50000
          mode = ncDIRECT
          edge_sw = ncPOSITIVE
          start_dir = ncPOSITIVE
          trigg_dir = ncPOSITIVE
          ref_pulse = ncOFF
          tr_s_block = 0
      basis:
        parameter:
          v_pos = 10000
          v_neg = 10000
          a1_pos = 50000
          a2_pos = 50000
          a1_neg = 50000
          a2_neg = 50000
    message:
      text:
        parameter:
          format = ncBREAK
          columns = 80
          data_modul = acp_err
```

### Program Logical/ConveyorBelt/conveyor (IEC) - Conveyor Logic Control

#### conveyorCyclic.ld - Cyclic code
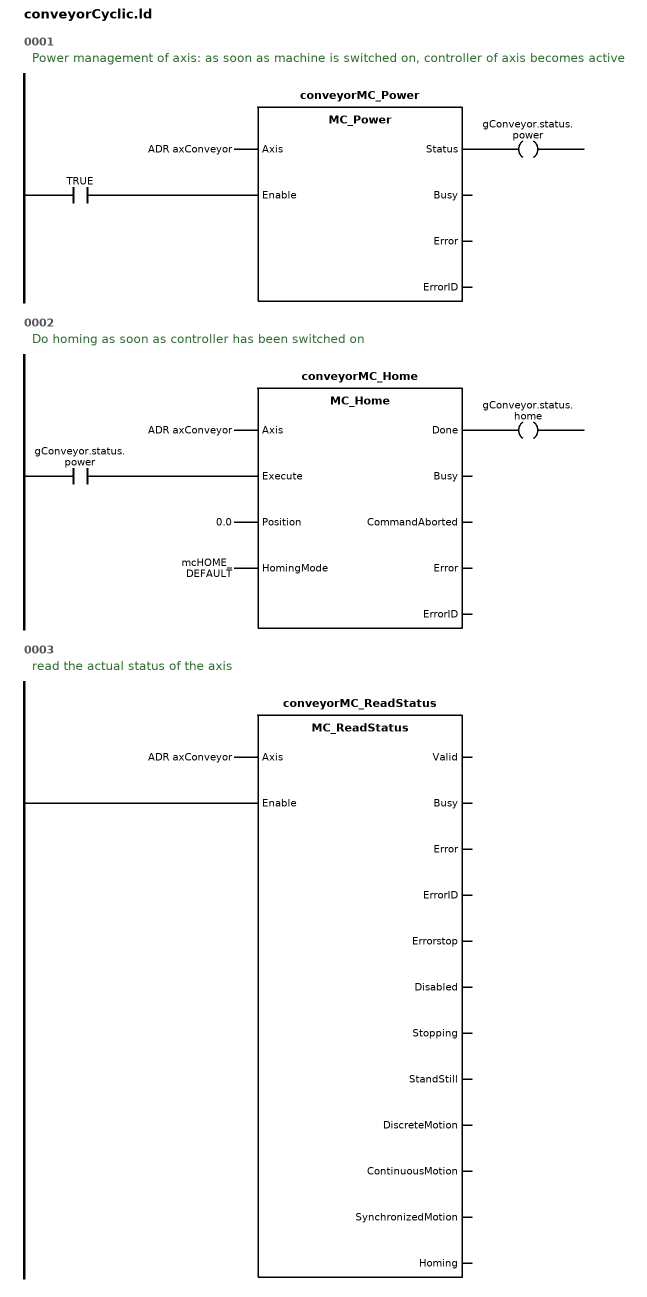
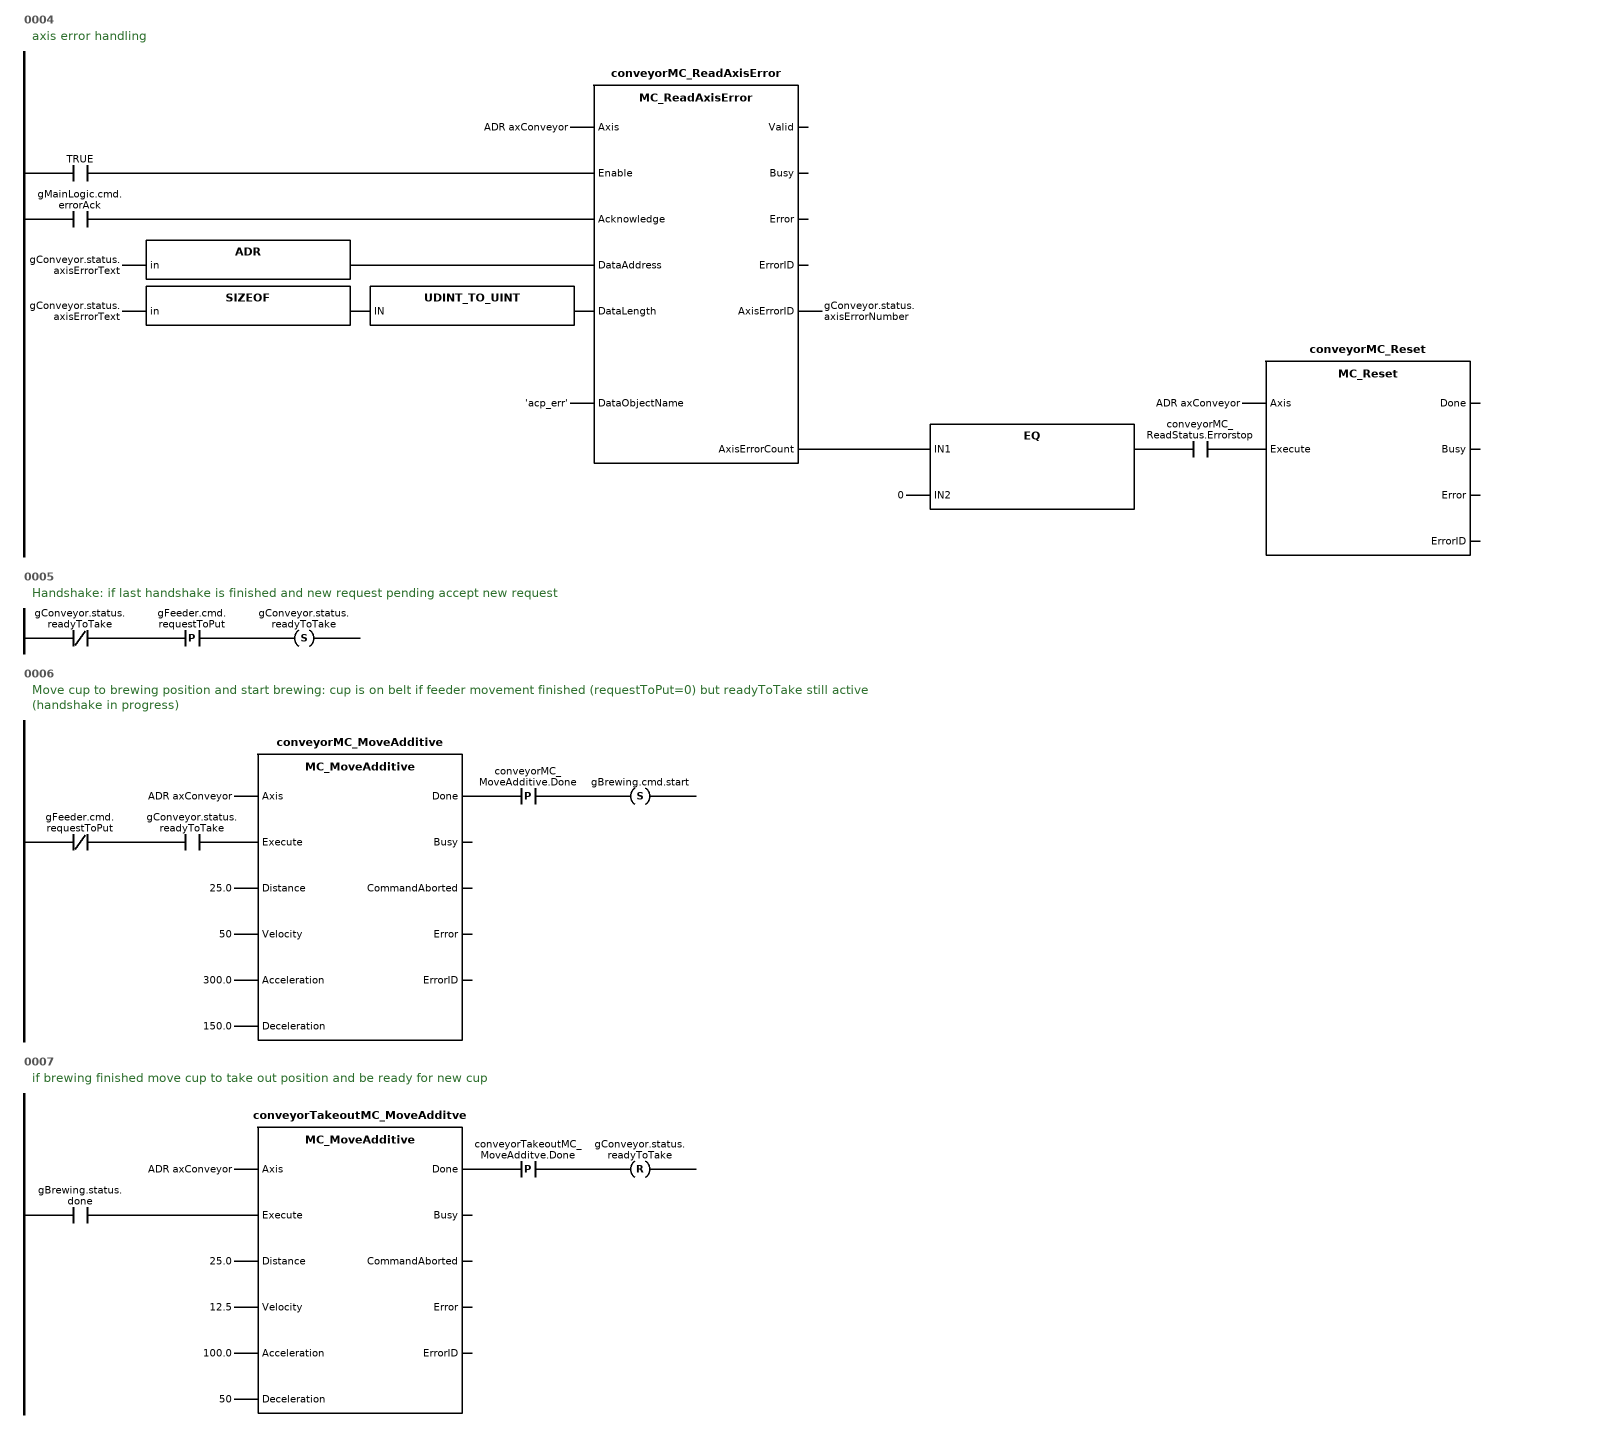
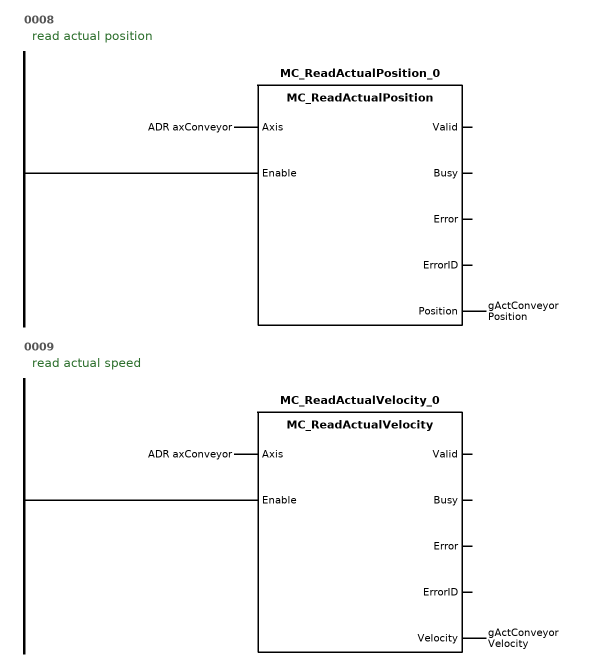
Ladder, written as Structured Text:
```iecst
(********************************************************************
 * COPYRIGHT -- Bernecker + Rainer
 ********************************************************************
 * Program: conveyor
 * File: conveyorCyclic.ld
 * Author: paulinw
 * Created: June 12, 2007
 ********************************************************************
 * Implementation of program conveyor
 ********************************************************************)

PROGRAM _CYCLIC
VAR
    _e1 : R_TRIG;
    _e2 : R_TRIG;
    _e3 : R_TRIG;
END_VAR
(* Network 1: Power management of axis: as soon as machine is switched on, controller of axis becomes active *)
conveyorMC_Power(Axis := ADR(axConveyor), Enable := TRUE);
gConveyor.status.power := conveyorMC_Power.Status;

(* Network 2: Do homing as soon as controller has been switched on *)
conveyorMC_Home(Axis := ADR(axConveyor), Execute := gConveyor.status.power, Position := 0.0, HomingMode := mcHOME_DEFAULT);
gConveyor.status.home := conveyorMC_Home.Done;

(* Network 3: read the actual status of the axis *)
conveyorMC_ReadStatus(Axis := ADR(axConveyor), Enable := TRUE);

(* Network 4: axis error handling *)
conveyorMC_ReadAxisError(Axis := ADR(axConveyor), Enable := TRUE, Acknowledge := gMainLogic.cmd.errorAck, DataAddress := ADR(in := gConveyor.status.axisErrorText), DataLength := UDINT_TO_UINT(SIZEOF(in := gConveyor.status.axisErrorText)), DataObjectName := 'acp_err');
gConveyor.status.axisErrorNumber := conveyorMC_ReadAxisError.AxisErrorID;
conveyorMC_Reset(Axis := ADR(axConveyor), Execute := (conveyorMC_ReadAxisError.AxisErrorCount = 0) AND conveyorMC_ReadStatus.Errorstop);

(* Network 5: Handshake: if last handshake is finished and new request pending accept new request *)
_e1(CLK := gFeeder.cmd.requestToPut);
IF NOT gConveyor.status.readyToTake AND _e1.Q THEN gConveyor.status.readyToTake := TRUE; END_IF;

(* Network 6: Move cup to brewing position and start brewing: cup is on belt if feeder movement finished (requestToPut=0) but readyToTake still active (handshake in progress) *)
conveyorMC_MoveAdditive(Axis := ADR(axConveyor), Execute := NOT gFeeder.cmd.requestToPut AND gConveyor.status.readyToTake, Distance := 25.0, Velocity := 50, Acceleration := 300.0, Deceleration := 150.0);
_e2(CLK := conveyorMC_MoveAdditive.Done);
IF conveyorMC_MoveAdditive.Done AND _e2.Q THEN gBrewing.cmd.start := TRUE; END_IF;

(* Network 7: if brewing finished move cup to take out position and be ready for new cup *)
conveyorTakeoutMC_MoveAdditve(Axis := ADR(axConveyor), Execute := gBrewing.status.done, Distance := 25.0, Velocity := 12.5, Acceleration := 100.0, Deceleration := 50);
_e3(CLK := conveyorTakeoutMC_MoveAdditve.Done);
IF conveyorTakeoutMC_MoveAdditve.Done AND _e3.Q THEN gConveyor.status.readyToTake := FALSE; END_IF;

(* Network 8: read actual position  *)
MC_ReadActualPosition_0(Axis := ADR(axConveyor), Enable := TRUE);
gActConveyorPosition := MC_ReadActualPosition_0.Position;

(* Network 9: read actual speed *)
MC_ReadActualVelocity_0(Axis := ADR(axConveyor), Enable := TRUE);
gActConveyorVelocity := MC_ReadActualVelocity_0.Velocity;
END_PROGRAM
```

### Package Logical/BrewingAssembly - Brewing & Dosing

### Program Logical/BrewingAssembly/brewing (IEC)

#### brewing.var - Local variables
```iecst
(********************************************************************
 * COPYRIGHT -- B&R
 ********************************************************************
 * Package: Brewing
 * File: brewing.var
 * Author: B&R
 * Created: June 14, 2007
 *******************************************************************)
VAR
	pBrewingText : UDINT := 0;
END_VAR
VAR CONSTANT
	sSTANDBY : UINT := 0;
	sDOSING : UINT := 10;
	sBREWING : UINT := 20;
	sFINISH : UINT := 30;
END_VAR
VAR
	milkTP : TP;
	coffeeTP : TP;
	sugarTP : TP;
	waterTP : TP;
END_VAR
```

### Package Logical/FeederArm - Feeder Control

### Data object Logical/FeederArm/acp_err (Ett)

- acp_err.ett (not shown)

- Data object Logical/FeederArm/feed_ini (Ax) (no source held here)

### Program Logical/FeederArm/feeder (IEC)

#### feederCyclic.ld - Cyclic code
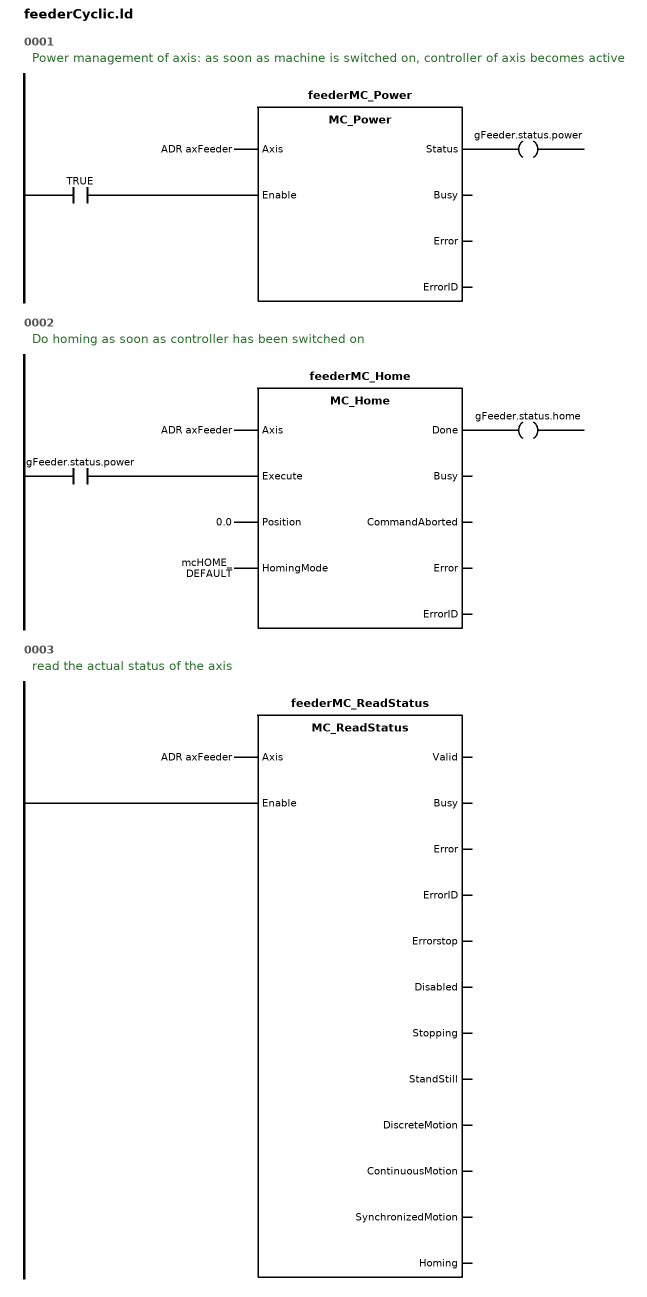
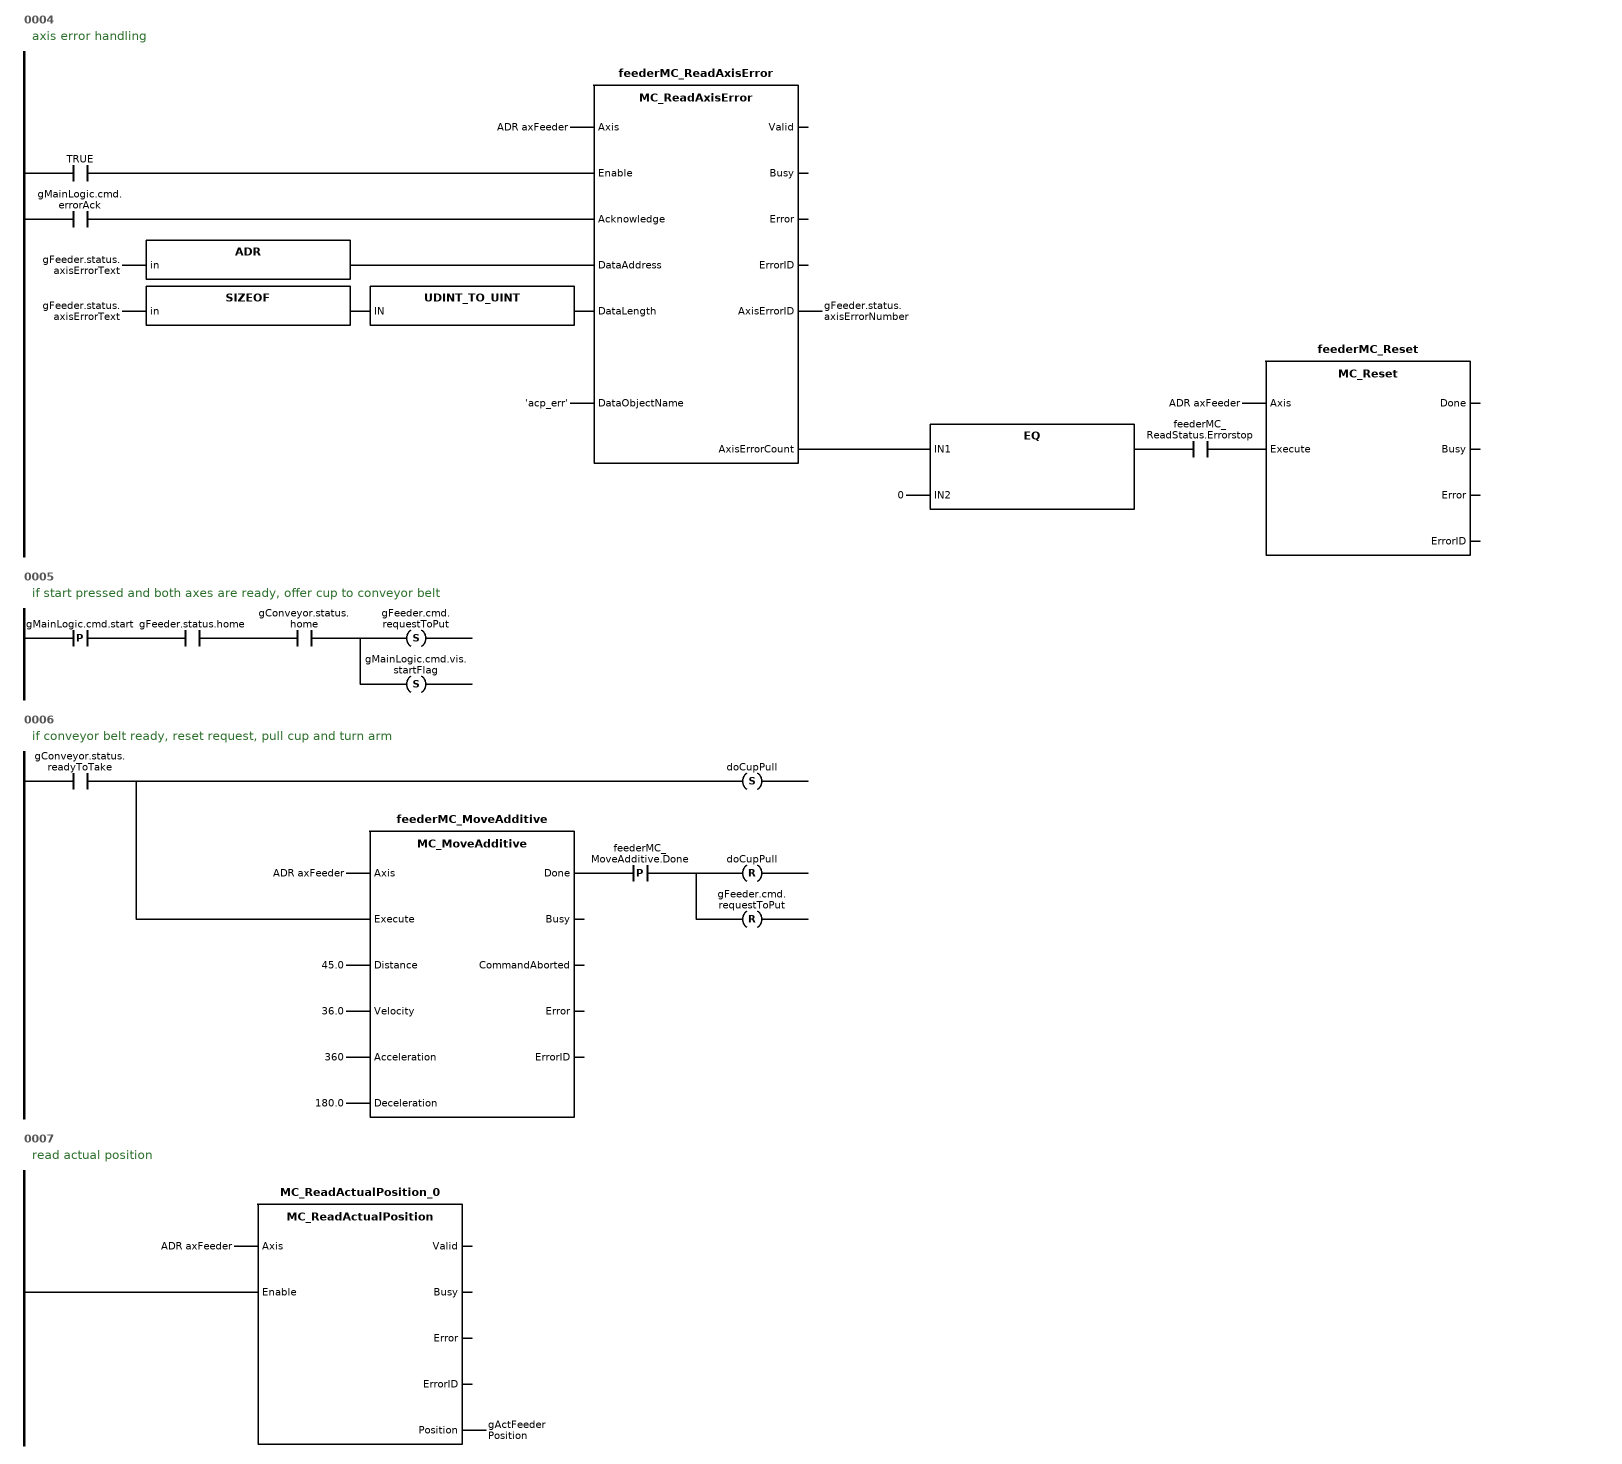
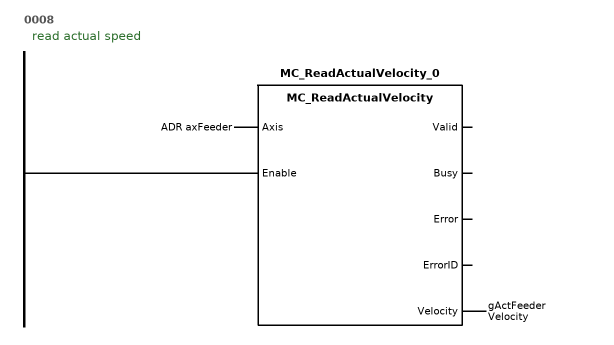
Ladder, written as Structured Text:
```iecst
(********************************************************************
 * COPYRIGHT -- Bernecker + Rainer
 ********************************************************************
 * Program: feeder
 * File: feederCyclic.ld
 * Author: paulinw
 * Created: June 13, 2007
 ********************************************************************
 * Implementation of program feeder
 ********************************************************************)

PROGRAM _CYCLIC
VAR
    _e1 : R_TRIG;
    _p2 : BOOL;
    _e3 : R_TRIG;
END_VAR
(* Network 1: Power management of axis: as soon as machine is switched on, controller of axis becomes active *)
feederMC_Power(Axis := ADR(axFeeder), Enable := TRUE);
gFeeder.status.power := feederMC_Power.Status;

(* Network 2: Do homing as soon as controller has been switched on  *)
feederMC_Home(Axis := ADR(axFeeder), Execute := gFeeder.status.power, Position := 0.0, HomingMode := mcHOME_DEFAULT);
gFeeder.status.home := feederMC_Home.Done;

(* Network 3: read the actual status of the axis *)
feederMC_ReadStatus(Axis := ADR(axFeeder), Enable := TRUE);

(* Network 4: axis error handling  *)
feederMC_ReadAxisError(Axis := ADR(axFeeder), Enable := TRUE, Acknowledge := gMainLogic.cmd.errorAck, DataAddress := ADR(in := gFeeder.status.axisErrorText), DataLength := UDINT_TO_UINT(SIZEOF(in := gFeeder.status.axisErrorText)), DataObjectName := 'acp_err');
gFeeder.status.axisErrorNumber := feederMC_ReadAxisError.AxisErrorID;
feederMC_Reset(Axis := ADR(axFeeder), Execute := (feederMC_ReadAxisError.AxisErrorCount = 0) AND feederMC_ReadStatus.Errorstop);

(* Network 5: if start pressed and both axes are ready, offer cup to conveyor belt *)
_e1(CLK := gMainLogic.cmd.start);
_p2 := _e1.Q AND gFeeder.status.home AND gConveyor.status.home;
IF _p2 THEN
    gFeeder.cmd.requestToPut := TRUE;
    gMainLogic.cmd.vis.startFlag := TRUE;
END_IF;

(* Network 6: if conveyor belt ready, reset request, pull cup and turn arm  *)
IF gConveyor.status.readyToTake THEN doCupPull := TRUE; END_IF;
feederMC_MoveAdditive(Axis := ADR(axFeeder), Execute := gConveyor.status.readyToTake, Distance := 45.0, Velocity := 36.0, Acceleration := 360, Deceleration := 180.0);
_e3(CLK := feederMC_MoveAdditive.Done);
IF feederMC_MoveAdditive.Done AND _e3.Q THEN
    doCupPull := FALSE;
    gFeeder.cmd.requestToPut := FALSE;
END_IF;

(* Network 7: read actual position  *)
MC_ReadActualPosition_0(Axis := ADR(axFeeder), Enable := TRUE);
gActFeederPosition := MC_ReadActualPosition_0.Position;

(* Network 8: read actual speed *)
MC_ReadActualVelocity_0(Axis := ADR(axFeeder), Enable := TRUE);
gActFeederVelocity := MC_ReadActualVelocity_0.Velocity;
END_PROGRAM
```

### Package Logical/FlowHeater - Heater Control

### Program Logical/FlowHeater/heating (ANSIC)

#### heating.var - Local variables
```iecst
(********************************************************************
 * COPYRIGHT -- B&R
 ********************************************************************
 * Package: heating
 * File: heating.var
 * Author: B&R
 * Created: June 15, 2007
 *******************************************************************)
VAR
	tempLCRPIDpara : LCRPIDpara := (0);
	tempLCRPID : LCRPID := (0);
	simLCRPT2 : LCRPT2 := (0);
END_VAR
```

### Package Logical/Recipes - Coffee Recipes

### Data object Logical/Recipes/regular (Simple) - Normal coffee

#### regular.dat
```
(********************************************************************
 * COPYRIGHT -- B&R
 ********************************************************************
 * Data object: regular
 * File: normal.dat
 * Author: B&R
 * Created: June 18, 2007
 ********************************************************************
 * Data object file: norma.dat
 ********************************************************************)
01.69	; price						[€]  - REAL
80.0	;	set temperature [°C] - REAL
100.0	; milk						[ml] - REAL
30.0	; sugar						[g]  - REAL
60.0  ; coffee powder		[g]  - REAL
150.0 ; water						[ml] - REAL
```

### Data object Logical/Recipes/cappu (Simple) - Cappucino

#### cappu.dat
```
(********************************************************************
 * COPYRIGHT -- B&R
 ********************************************************************
 * Data object: cappu
 * File: cappu.dat
 * Author: B&R
 * Created: June 18, 2007
 ********************************************************************
 * Data object file: cappu.dat
 ********************************************************************)
01.39	; price						[€]  - REAL
70.0	;	set temperature [°C] - REAL
200.0	; milk						[ml] - REAL
60.0	; sugar						[g]  - REAL
60.0  ; coffee powder		[g]  - REAL
150.0 ; water						[ml] - REAL
```

### Data object Logical/Recipes/espres (Simple) - Espresso

#### espres.dat
```
(********************************************************************
 * COPYRIGHT -- B&R
 ********************************************************************
 * Data object: espress
 * File: espress.dat
 * Author: B&R
 * Created: June 18, 2007
 ********************************************************************
 * Data object file: espres.dat
 ********************************************************************)
01.55	; price						[€]  - REAL
92.0	;	set temperature [°C] - REAL
00.0	; milk						[ml] - REAL
20.0	; sugar						[g]  - REAL
80.0  ; coffee powder		[g]  - REAL
50.0  ; water						[ml] - REAL
```

- Visualisation Logical/Visualisation (not shown)

### Package Logical/Libraries - Global Libraries

### Library Logical/Libraries/CoffeeLib (IEC)

#### CoffeeLib.fun - Exported functions and function blocks
```iecst
(********************************************************************
 * COPYRIGHT -- B&R
 ********************************************************************
 * Library: CoffeeLib
 * File: CoffeeLib.fun
 * Author: B&R
 * Created: June 18, 2007
 ********************************************************************
 * Functions and function blocks of library CoffeeLib
 ********************************************************************)

FUNCTION_BLOCK MoneyChanger (*Changes given money based on euros*)
	VAR_INPUT
		execute : BOOL; (*Do change*)
		given : REAL; (*Given money*)
		price : REAL; (*Price*)
	END_VAR
	VAR_OUTPUT
		change : REAL; (*total money to change*)
		cent1 : USINT; (*Number of 1 Cent coins*)
		cent2 : USINT; (*Number of 2 Cent coins*)
		cent5 : USINT; (*Number of 5 Cent coins*)
		cent10 : USINT; (*Number of 10 Cent coins*)
		cent20 : USINT; (*Number of 20 Cent coins*)
		cent50 : USINT; (*Number of 50 Cent coins*)
		euro1 : UDINT; (*Number of 1 Euro coins*)
		euro2 : UDINT; (*Number of 2 Euro coins*)
		resetMoney : REAL; (*Resets given money*)
	END_VAR
	VAR
		centChange : USINT; (*cent change calculation*)
		executeOld : BOOL; (*edge sensitive operation*)
	END_VAR
END_FUNCTION_BLOCK
```

### Program Logical/NewProgram (IEC) - Program

#### NewProgram.st - Implementation code
```iecst
(********************************************************************
 * COPYRIGHT -- B&R Industrial Automation GmbH
 ********************************************************************
 * Program: NewProgram
 * File: NewProgram.st
 * Author: hilchenbachc
 * Created: October 28, 2022
 ********************************************************************
 * Implementation of program NewProgram
 ********************************************************************)

PROGRAM _INIT

timedelta := T#-3s;

_mystruct.a_bool := TRUE;
_mystruct.text1 := "Unicode";
_mystruct.text2 := 'ASCII';

FOR n := 0 TO 9 DO
	_mystruct.inner1.an_int_array[n] := -5-n;
END_FOR

_mystruct.an_int := -3;
_mystruct.inner1.inner2.an_usint := 7;
_mystruct.inner1.inner2.an_usint := 9;
_mystruct.inner1.inner2.inner3.an_usint := 11;
_mystruct.inner1.inner2.inner3.ton.PT := T#34ms;

//FOR n := 0 TO 9 DO
//	myStructArray[n] := _mystruct;
//	myStructArray[n].an_int := -11-n;
//	myStructArray[n].inner1.inner2.an_usint := INT_TO_USINT(n);
//END_FOR

 sizeofmystruct := SIZEOF(_mystruct);

//floatarray[0] := 3.14;

END_PROGRAM

PROGRAM _CYCLIC

_mystruct.ton( PT := T#4s56ms, IN := TRUE );

END_PROGRAM
```

#### variable.var - Local variables
```iecst
(********************************************************************
 * COPYRIGHT -- B&R Industrial Automation GmbH
 ********************************************************************
 * Program: NewProgram
 * File: variable.var
 * Author: hilchenbachc
 * Created: October 28, 2022
 ********************************************************************
 * Local variables of program NewProgram
 ********************************************************************)
VAR
	timedelta : TIME := T#0S;
	n : INT := 0; (*myStructArray : ARRAY[0..9] OF MyStruct := [10(0)];*) (*floatarray : ARRAY[0..2] OF REAL;*)
	sizeofmystruct : UDINT := 0;
	_mystruct : MyStruct := (0);
END_VAR
```

#### Types.typ - Local data types
```iecst
(********************************************************************
 * COPYRIGHT -- B&R Industrial Automation GmbH
 ********************************************************************
 * Program: NewProgram
 * File: Types.typ
 * Author: hilchenbachc
 * Created: October 31, 2022
 ********************************************************************
 * Local data types of program NewProgram
 ********************************************************************)

TYPE
	InnerInnerInnerStruct : 	STRUCT
		an_usint : USINT;
		ton : TON := (PT:=T#1234ms);
	END_STRUCT;
	InnerInnerStruct : 	STRUCT
		an_usint : USINT;
		inner3 : InnerInnerInnerStruct;
	END_STRUCT;
	InnerStruct : 	STRUCT
		an_int_array : ARRAY[0..9]OF INT;
		inner2 : InnerInnerStruct;
	END_STRUCT;
	MyStruct : 	STRUCT
		a_bool : BOOL;
		ton : TON;
		text1 : WSTRING[13];
		text2 : STRING[13];
		inner1 : InnerStruct;
		an_int : INT;
	END_STRUCT;
END_TYPE
```

### Program Logical/myProg (IEC) - Program

#### myProg.st - Implementation code
```iecst
(********************************************************************
 * COPYRIGHT -- B&R Industrial Automation GmbH
 ********************************************************************
 * Program: myProg
 * File: myProg.st
 * Author: hilchenbachc
 * Created: November 22, 2022
 ********************************************************************
 * Implementation of program myProg
 ********************************************************************)

PROGRAM _INIT
	myUSINT;
	myUINT;
	mySTRING;
	myWSTRING;
	myTIME;
	myTOD;
	myDT;
	myDINT;
	myINTArray;
	mySTRINGArray;
	myUDINT;
	myDATE;
	myLREAL;
	myREAL;
	myINT;
	mySINT;
	myBOOL;
	myREALArray;
END_PROGRAM

PROGRAM _CYCLIC

END_PROGRAM
```

#### myProg.var - Local variables
```iecst
(********************************************************************
 * COPYRIGHT -- B&R Industrial Automation GmbH
 ********************************************************************
 * Program: myProg
 * File: myProg.var
 * Author: hilchenbachc
 * Created: November 22, 2022
 ********************************************************************
 * Local variables of program myProg
 ********************************************************************)
VAR
	myREALArray : ARRAY[0..9] OF REAL := [10(0.0)];
	myUSINT : USINT := 0;
	myUINT : UINT := 0;
	mySTRING : STRING[80] := '';
	myWSTRING : WSTRING[80] := "";
	myTIME : TIME := T#0S;
	myTOD : TIME_OF_DAY := TOD#00:00:00;
	myDT : DATE_AND_TIME := DT#1970-01-01-00:00:00;
	myDINT : DINT := 0;
	myINTArray : ARRAY[0..9] OF INT := [10(0)];
	mySTRINGArray : ARRAY[0..9] OF STRING[80] := [''];
	myUDINT : UDINT := 0;
	myDATE : DATE;
	myLREAL : LREAL := 0.0;
	myREAL : REAL := 0.0;
	myINT : INT := 0;
	mySINT : SINT := 0;
	myBOOL : BOOL := FALSE;
END_VAR
```

#### Type.typ - not listed in the package file held
```iecst
TYPE
	myStructType2 : 	STRUCT
		struct1 : myStructType;
		structList : ARRAY[0..2]OF myStructType;
	END_STRUCT;
	myStructType : 	STRUCT
		member1 : USINT := 3;
		member2 : ARRAY[0..2]OF USINT := [33,44,55];
	END_STRUCT;
	myEnumType :
		(
		eins,
		zwei,
		drei
		);
	myDerivedType1 :USINT(4..6) ;
	myDerivedType2 :ARRAY[3..6]OF USINT;
	myComplexStructType : 	STRUCT
		bool : BOOL;
		usint : USINT;
		uint : UINT;
		udint : UDINT;
		sint : SINT;
		int : INT;
		dint : DINT;
		real : REAL;
		lreal : LREAL;
		time : TIME;
		tod : TIME_OF_DAY;
		date : DATE;
		dt : DATE_AND_TIME;
		string : STRING[80];
		wstring : WSTRING[80];
		stringlist : ARRAY[1..10]OF STRING[40] := ['A','B','C','D','E','F','G','H','I','J'];
		wstringlist : ARRAY[1..10]OF WSTRING[40] := ["A","B","C","D","E","F","G","H","I","J"];
		vector : ARRAY[1..10]OF REAL;
		intvector : ARRAY[0..9]OF INT;
		intvector2 : ARRAY[0..0]OF INT;
		matrix : ARRAY[0..9,0..3]OF REAL;
		myStruct0 : myStructType;
		myStruct1 : ARRAY[0..1]OF myStructType;
		myStruct2 : ARRAY[2..2]OF myStructType;
		myStruct3 : ARRAY[-1..1]OF myStructType;
		myStruct4 : ARRAY[0..2,0..3]OF myStructType;
		myStruct5 : ARRAY[0..2]OF myStructType2;
		myStruct6 : ARRAY[1..2,-1..1]OF myStructType2;
		myEnum : myEnumType;
		enumlist : ARRAY[0..4]OF myEnumType;
		enumlist2 : ARRAY[0..0]OF myEnumType;
		subrange1 : SINT(-3..6) ;
		derived1 : myDerivedType1;
		derived2 : myDerivedType2;
		n : USINT := 99;
	END_STRUCT;
END_TYPE
```

- Data object Logical/cnc3 (Cnc) - CNC Program (no source held here)

### Data object Logical/data (Simple) - Simple data object

#### data.dat
```
(********************************************************************
 * COPYRIGHT -- B&R Industrial Automation GmbH
 ********************************************************************
 * Data object: data
 * File: data.dat
 * Author: hilchenbachc
 * Created: April 18, 2023
 ********************************************************************
 * Data object file: data.dat
 ********************************************************************)
'A'
```

Listed in the project but not available here: Logical/Doc, Logical/Global.typ, Logical/ConveyorBelt/conveyor/conveyor.var, Logical/BrewingAssembly/brewing/brewing.st, Logical/FeederArm/feeder/feeder.var, Logical/FlowHeater/heating/heating.c, Logical/Recipes/empty1, Logical/Recipes/object2, Logical/Libraries/CoffeeLib/CoffeeLib.st, Logical/cnc1, Logical/cnc2
